Xinje XDPPro project, PLC1: XL3-16 (software 3.7.17c 2024-04-02)

PROGRAM Ladder

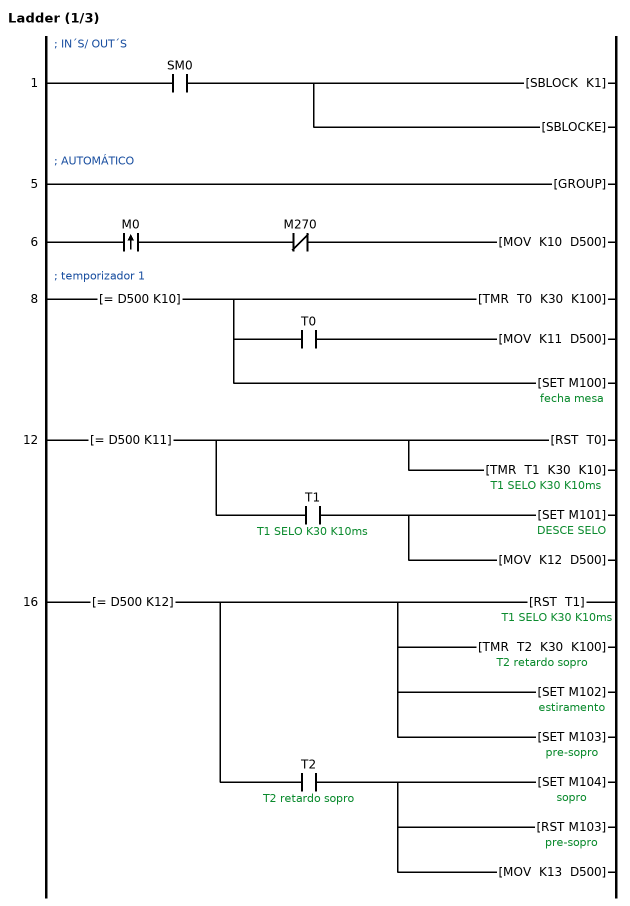
; IN´S/ OUT´S 
LD     SM0
SBLOCK K1
SBLOCKE
; AUTOMÁTICO
GROUP
LDP    M0
ANI    M270
MOV    K10 D500
; temporizador 1
LD=    D500 K10
TMR    T0 K30 K100
MPS
AND    T0
MOV    K11 D500
MPP
SET    M100	; fecha mesa
LD=    D500 K11
RST    T0
TMR    T1 K30 K10	; T1 SELO K30 K10ms
AND    T1	; T1 SELO K30 K10ms
SET    M101	; DESCE SELO
MOV    K12 D500
LD=    D500 K12
RST    T1	; T1 SELO K30 K10ms
TMR    T2 K30 K100	; T2 retardo sopro
SET    M102	; estiramento
SET    M103	; pre-sopro
AND    T2	; T2 retardo sopro
SET    M104	; sopro
RST    M103	; pre-sopro
MOV    K13 D500

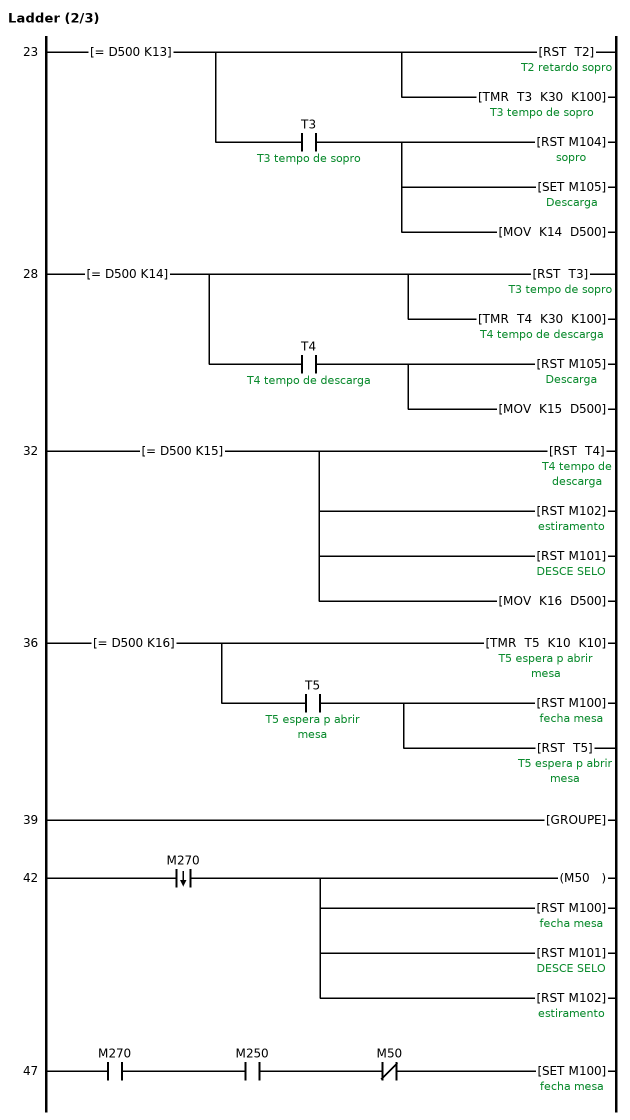
LD=    D500 K13
RST    T2	; T2 retardo sopro
TMR    T3 K30 K100	; T3 tempo de sopro
AND    T3	; T3 tempo de sopro
RST    M104	; sopro
SET    M105	; Descarga
MOV    K14 D500
LD=    D500 K14
RST    T3	; T3 tempo de sopro
TMR    T4 K30 K100	; T4 tempo de descarga
AND    T4	; T4 tempo de descarga
RST    M105	; Descarga
MOV    K15 D500
LD=    D500 K15
RST    T4	; T4 tempo de descarga
RST    M102	; estiramento
RST    M101	; DESCE SELO
MOV    K16 D500
LD=    D500 K16
TMR    T5 K10 K10	; T5 espera p abrir mesa
AND    T5	; T5 espera p abrir mesa
RST    M100	; fecha mesa
RST    T5	; T5 espera p abrir mesa
GROUPE
LDF    M270
OUT    M50
RST    M100	; fecha mesa
RST    M101	; DESCE SELO
RST    M102	; estiramento
LD     M270
AND    M250
ANI    M50
SET    M100	; fecha mesa

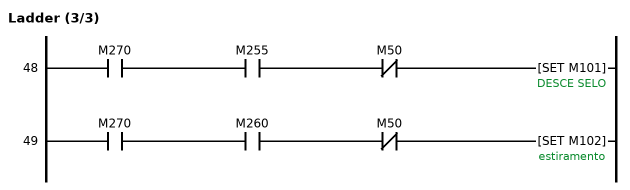
LD     M270
AND    M255
ANI    M50
SET    M101	; DESCE SELO
LD     M270
AND    M260
ANI    M50
SET    M102	; estiramento

COMMENTS (devices not used above)
X1	EMERGENCIA
Y0	PUL- MOTOR DE PASSO
Y2	DIR - NOTOR DE PASSO
Y7	FACA
Y4	ENA - MOTOR DE PASSO
X6	SENSOR FACA CIMA
M6	SENSOR FACA CIMA
M1	EMERGENCIA
M107	FACA
HD100	Ø_Rolo_Puxador_IHM
HD102	PI (3,141592)
HD0	Distancia_Puxador_IHM
HD2	Freq_%_IHM
D102	Freq_Hz
D100	Pulse
X4	ON
M4	ON
M5	SENSOR FACA BAIXO
X5	SENSOR FACA BAIXO

SBLOCK K1	; In's/Out's
  ; In's/Out's
  ;ENTRADAS
  LD X0
  OUT M0
  LD X1
  OUT M1
  LD X2
  OUT M2
  LD X3
  OUT M3
  LD X4
  OUT M4
  LDI X5
  OUT M5
  LD X6
  OUT M6
  LD X7
  OUT M7
  LD X10
  OUT M10
  LD X11
  OUT M11
  LD X12
  OUT M12
  LD X13
  OUT M13
  LD X14
  OUT M14
  LD X15
  OUT M15
  LD X16
  OUT M16
  LD X17
  OUT M17
  ;SAÍDAS
  LD M100
  OUT Y0
  LD           M101
  OUT        Y1
  LD           M102
  OUT        Y2
  LD M103
  OUT Y3
  LD M104
  OUT Y4
  LD M105
  OUT Y5
  LD M106
  OUT Y6
  LD M107
  OUT Y7
  LD M110
  OUT Y10
  LD M111
  OUT Y11